(* PLC project BlogProject.project, CODESYS CODESYS V3.5 SP14 Patch 3 *)
(* stored: creationDateTime 2021-10-07T21:02:08.3158574, modificationDateTime 2021-10-07T20:40:20.1109198 *)

(* values of enumState: SYSTEM_OFF: Система выключена; SYSTEM_CHECK: Проверка сиситемы; SYSTEM_START: Старт системы; SYSTEM_RUN: Cистема в работе; SYSTEM_STOP: Остановка системы; SYSTEM_ERR: Ошибка системы *)

{attribute 'qualified_only'}
{attribute 'strict'}
TYPE enumState : (SYSTEM_OFF := 0, SYSTEM_CHECK := 1, SYSTEM_START := 2, SYSTEM_RUN := 3, SYSTEM_STOP := 4, SYSTEM_ERR := 5);
END_TYPE
